TYPE stSktPara :
STRUCT
	AutoReconnect : BOOL;
	EnableSendLog : BOOL;
	EnableRecvLog : BOOL;
	SendRecvTimeOut : TIME := T#3S;
	
END_STRUCT
END_TYPE

(* stored: Version 1.1.0.1, ProductVersion 3.1.4024.12
   DUT stSktPara: Id {ca22775b-3b46-4f09-a564-b5375d452e61} *)
